            $ 635 "A_sel_v≔A_VL1"
            global A_sel_v=A_VL1
            $ 636 "A_sel_v_end≔A_VL1_END"
            global A_sel_v_end=A_VL1_END
            $ 637 "b2_par_cd≔0"
            global b2_par_cd=0
            $ 638 "If b1_cell_info_L≟A or b1_cell_info_L≟C or b1_cell_info_L≟c"
            if (b1_cell_info_L == A  or  b1_cell_info_L == C  or  b1_cell_info_L == c):
              $ 639 "Scallup_check≔ True "
              global Scallup_check=  True
            else:
              $ 640 "Else" "noBreak"
              $ 641 "Scallup_check≔ False "
              global Scallup_check=  False
            end
            $ 642 "Call MoveandTouchFun_3f"
            MoveandTouchFun_3f()
            $ 643 "If b1_cell_info_L≟A or b1_cell_info_L≟C or b1_cell_info_L≟c"
            if (b1_cell_info_L == A  or  b1_cell_info_L == C  or  b1_cell_info_L == c):
              $ 644 "If A_Prepos_l[A_HOR]≟p[0,0,0,0,0,0]"
              if (A_Prepos_l[A_HOR] == p[0,0,0,0,0,0]):
                $ 645 "direction(p[0,0,0,0,0,0],[0,-1,0],8,120,160)"
                direction(p[0,0,0,0,0,0],[0,-1,0],8,120,160)
                $ 647 "AAgcp≔get_actual_tcp_pose()"
                global AAgcp= get_actual_tcp_pose ()
                $ 648 "AAgangle≔up_left"
                global AAgangle=p[.492775857339, .409517380626, -.029063830209, -2.419264859926, -.998084331190, -1.368689080860]
                $ 649 "AAgtp≔p[AAgcp[0],AAgcp[1],AAgcp[2],AAgangle[3],AAgangle[4],AAgangle[5]]"
                global AAgtp=p[AAgcp[0],AAgcp[1],AAgcp[2],AAgangle[3],AAgangle[4],AAgangle[5]]
                $ 650 "MoveL"
                $ 651 "AAgtp" "breakAfter"
                movel(pose_trans(Base, AAgtp), a=0.08, v=0.08)
                $ 653 "for_z_VL1≔contact_fun(p[0,0,0,0,0,0],[0,0,-1],10000,15,15,  False)"
                global for_z_VL1=contact_fun(p[0,0,0,0,0,0],[0,0,-1],10000,15,15,  False)
                $ 654 "direction(p[0,0,0,0,0,0],[0,0,1],20,120,160)"
                direction(p[0,0,0,0,0,0],[0,0,1],20,120,160)
                $ 655 "write_welder(4, False )"
                write_welder(4,  False  )
              else:
                $ 656 "Else" "noBreak"
                $ 657 "for_z_VL1≔p[0,0,0,0,0,0]"
                global for_z_VL1=p[0,0,0,0,0,0]
              end
            end
            $ 658 "If top_touch_3f"
            if (top_touch_3f):
              $ 659 "touch_3f_up"
              $ 660 "b_touch_pos≔pose_add(A_Prepos_l[A_VL1], p[0,0,a8_wv_distance/1000,0,0,0])"
              global b_touch_pos= pose_add (A_Prepos_l[A_VL1], p[0,0,a8_wv_distance/1000,0,0,0])
              $ 661 "b_touch_pos≔tilt_3f_fun(b_touch_pos,[0,0],a5_f_hole[1])"
              global b_touch_pos=tilt_3f_fun(b_touch_pos,[0,0],a5_f_hole[1])
              $ 662 "MoveL"
              $ 663 "b_touch_pos" "breakAfter"
              movel(pose_trans(Base, b_touch_pos), a=0.35, v=0.35)
              $ 664 "touch_result≔touch_fun2(b_touch_pos,b2_left_par,b9_touch_sens)"
              global touch_result=touch_fun2(b_touch_pos,b2_left_par,b9_touch_sens)
              $ 665 "A_Touch_p[A_sel_v_end]=touch_result"
              A_Touch_p[A_sel_v_end]=touch_result
              $ 666 "If EXT_flag1[3]≟ True "
              if (EXT_flag1[3] ==   True  ):
                $ 667 "MoveL"
                $ 668 "manual_tp≔A_Touch_p[A_sel_v_end]"
                global manual_tp=A_Touch_p[A_sel_v_end]
                $ 669 "manual_tp≔tilt_3f_fun(A_Touch_p[A_sel_v_end],basic_tilt_3f,0)"
                global manual_tp=tilt_3f_fun(A_Touch_p[A_sel_v_end],basic_tilt_3f,0)
                $ 670 "manual_tp≔pose_trans(manual_tp, p[0,0,-10/1000,0,0,0])"
                global manual_tp= pose_trans (manual_tp, p[0,0,-10/1000,0,0,0])
                $ 671 "manual_tp" "breakAfter"
                movel(pose_trans(Base, manual_tp), a=0.3, v=0.15)
                $ 672 "Wait: 1.5"
                sleep(1.5)
              end
            end
          end
          $ 673 "HOR_ML"
          $ 674 "If A_Prepos_l[A_HOR_ML]≠p[0,0,0,0,0,0]"
          if (A_Prepos_l[A_HOR_ML] != p[0,0,0,0,0,0]):
            $ 675 "b2_left_par≔ True "
            global b2_left_par=  True
            $ 676 "b8_wv_2f≔ True "
            global b8_wv_2f=  True
            $ 677 "b7_tilt_degree≔[0,0,0]"
            global b7_tilt_degree=[0,0,0]
            $ 678 "A_sel_v≔A_HOR_ML"
            global A_sel_v=A_HOR_ML
            $ 679 "If b1_cell_info_L≟C or b1_cell_info_L≟D"
            if (b1_cell_info_L == C  or  b1_cell_info_L == D):
              $ 680 "wv_direction≔1"
              global wv_direction=1
              $ 681 "Call MoveFun"
              MoveFun()
              $ 682 "for_cal_xy≔contact_fun(p[0,0,0,0,0,0],[1,0,0],20000,20,20)"
              global for_cal_xy=contact_fun(p[0,0,0,0,0,0],[1,0,0],20000,20,20)
              $ 683 "direction(p[0,0,0,0,0,0],[-1,0,0],15,120,160)"
              direction(p[0,0,0,0,0,0],[-1,0,0],15,120,160)
              $ 684 "direction(p[0,0,0,0,0,0],[0,-1,0],60,120,160)"
              direction(p[0,0,0,0,0,0],[0,-1,0],60,120,160)
              $ 685 "direction(p[0,0,0,0,0,0],[1,0,0],20,120,160)"
              direction(p[0,0,0,0,0,0],[1,0,0],20,120,160)
              $ 686 "for_cal_x_wel≔contact_fun(p[0,0,0,0,0,0],[0,1,0],20000,20,20)"
              global for_cal_x_wel=contact_fun(p[0,0,0,0,0,0],[0,1,0],20000,20,20)
              $ 687 "direction(p[0,0,0,0,0,0],[0,-1,0],20,120,160)"
              direction(p[0,0,0,0,0,0],[0,-1,0],20,120,160)
              $ 688 "for_cal_y_wel≔contact_fun(p[0,0,0,0,0,0],[1,0,0],20000,20,20)"
              global for_cal_y_wel=contact_fun(p[0,0,0,0,0,0],[1,0,0],20000,20,20)
              $ 689 "direction(p[0,0,0,0,0,0],[-1,0,0],20,120,160)"
              direction(p[0,0,0,0,0,0],[-1,0,0],20,120,160)
              $ 690 "for_z_VLR2≔contact_fun(p[0,0,0,0,0,0],[0,0,-1],20000,20,20)"
              global for_z_VLR2=contact_fun(p[0,0,0,0,0,0],[0,0,-1],20000,20,20)
              $ 691 "direction(p[0,0,0,0,0,0],[0,0,1],20,120,160)"
              direction(p[0,0,0,0,0,0],[0,0,1],20,120,160)
              $ 692 "for_cal_rot≔A_Touch_p[A_HOR]"
              global for_cal_rot=A_Touch_p[A_HOR]
              $ 693 "A_Touch_p[A_sel_v]=p[for_cal_xy[0],for_cal_xy[1],for_z_VLR2[2],for_cal_rot[3],for_cal_rot[4],for_cal_rot[5]]"
              A_Touch_p[A_sel_v]=p[for_cal_xy[0],for_cal_xy[1],for_z_VLR2[2],for_cal_rot[3],for_cal_rot[4],for_cal_rot[5]]
              $ 694 "A_Touch_p[A_sel_v]=pose_trans(A_Touch_p[A_sel_v], p[Touch_dis/1000,0,0,0,0,0])"
              A_Touch_p[A_sel_v]= pose_trans (A_Touch_p[A_sel_v], p[Touch_dis/1000,0,0,0,0,0])
              $ 695 "write_welder(4, False )"
              write_welder(4,  False  )
            else:
              $ 696 "Else" "noBreak"
              $ 697 "wv_direction≔1"
              global wv_direction=1
              $ 698 "for_cal_rot≔A_Touch_p[A_HOR]"
              global for_cal_rot=A_Touch_p[A_HOR]
              $ 699 "Call MoveFun_cd"
              MoveFun_cd()
              $ 700 "for_cal_y_wel≔contact_fun(p[0,0,0,0,0,0],[1,0,0],20000,20,20)"
              global for_cal_y_wel=contact_fun(p[0,0,0,0,0,0],[1,0,0],20000,20,20)
              $ 701 "for_cal_y_wel[2]=for_cal_rot[2]"
              for_cal_y_wel[2]=for_cal_rot[2]
              $ 702 "dir_x_cal≔get_feature_Line(for_cal_rot,for_cal_y_wel)"
              global dir_x_cal=get_feature_Line(for_cal_rot,for_cal_y_wel)
              $ 703 "direction(p[0,0,0,0,0,0],[-1,0,0],40,120,160)"
              direction(p[0,0,0,0,0,0],[-1,0,0],40,120,160)
              $ 704 "direction(p[0,0,0,0,0,0],[0,-1,0],80,120,160)"
              direction(p[0,0,0,0,0,0],[0,-1,0],80,120,160)
              $ 705 "for_cal_y_wel≔contact_fun(p[0,0,0,0,0,0],[1,0,0],20000,20,20)"
              global for_cal_y_wel=contact_fun(p[0,0,0,0,0,0],[1,0,0],20000,20,20)
              $ 706 "direction(p[0,0,0,0,0,0],[-1,0,0],5,120,160)"
              direction(p[0,0,0,0,0,0],[-1,0,0],5,120,160)
              $ 707 "direction(p[0,0,0,0,0,0],[0,1,0],60,120,160)"
              direction(p[0,0,0,0,0,0],[0,1,0],60,120,160)
              $ 708 "direction(p[0,0,0,0,0,0],[1,0,0],7,120,160)"
              direction(p[0,0,0,0,0,0],[1,0,0],7,120,160)
              $ 709 "for_cal_x_wel≔contact_fun(p[0,0,0,0,0,0],[0,-1,0],20000,20,20)"
              global for_cal_x_wel=contact_fun(p[0,0,0,0,0,0],[0,-1,0],20000,20,20)
              $ 710 "get_ml≔get_feature_pose(for_cal_x_wel,for_cal_rot)"
              global get_ml=get_feature_pose(for_cal_x_wel,for_cal_rot)
              $ 712 "A_Touch_p[A_sel_v]=feature_offset(for_cal_rot,p[0,get_ml[0]+(-cd_offset+cd_extra_dis)/1000,0,0,0,0],dir_x_cal)"
              A_Touch_p[A_sel_v]=feature_offset(for_cal_rot,p[0,get_ml[0]+(-cd_offset+cd_extra_dis)/1000,0,0,0,0],dir_x_cal)
              $ 713 "direction(p[0,0,0,0,0,0],[0,1,0],5,120,160)"
              direction(p[0,0,0,0,0,0],[0,1,0],5,120,160)
              $ 714 "direction(p[0,0,0,0,0,0],[-1,0,0],20,120,160)"
              direction(p[0,0,0,0,0,0],[-1,0,0],20,120,160)
              $ 715 "write_welder(4, False )"
              write_welder(4,  False  )
            end
            $ 716 "homeing()"
            homeing()
          else:
            $ 717 "Else" "noBreak"
            $ 718 "homeing()"
            homeing()
          end
          $ 719 "VL2"
          $ 720 "If A_Prepos_l[A_VL2]≠p[0,0,0,0,0,0]"
          if (A_Prepos_l[A_VL2] != p[0,0,0,0,0,0]):
            $ 721 "b2_left_par≔ True "
            global b2_left_par=  True
            $ 722 "b8_wv_2f≔ False "
            global b8_wv_2f=  False
            $ 723 "b7_tilt_degree≔basic_tilt_3f"
            global b7_tilt_degree=basic_tilt_3f
            $ 724 "A_sel_v≔A_VL2"
            global A_sel_v=A_VL2
            $ 725 "A_sel_v_end≔A_VL2_END"
            global A_sel_v_end=A_VL2_END
            $ 726 "b2_par_cd≔1"
            global b2_par_cd=1
            $ 727 "If b1_cell_info_L≟A or b1_cell_info_L≟C or b1_cell_info_L≟c"
            if (b1_cell_info_L == A  or  b1_cell_info_L == C  or  b1_cell_info_L == c):
              $ 728 "Scallup_check≔ True "
              global Scallup_check=  True
            else:
              $ 729 "Else" "noBreak"
              $ 730 "Scallup_check≔ False "
              global Scallup_check=  False
            end
            $ 731 "If b1_cell_info_L≟d or b1_cell_info_L≟c"
            if (b1_cell_info_L == d  or  b1_cell_info_L == c):
              $ 732 "Halt"
              halt
            else:
              $ 733 "Else" "noBreak"
              $ 734 "If A_Touch_p[A_VL1]≟p[0,0,0,0,0,0]"
              if (A_Touch_p[A_VL1] == p[0,0,0,0,0,0]):
                $ 735 "Call MoveandTouchFun_3f"
                MoveandTouchFun_3f()
                $ 736 "If A_Prepos_l[A_HOR_ML]≟p[0,0,0,0,0,0]"
                if (A_Prepos_l[A_HOR_ML] == p[0,0,0,0,0,0]):
                  $ 737 "direction(p[0,0,0,0,0,0],[-1,-1,0],8,120,160)"
                  direction(p[0,0,0,0,0,0],[-1,-1,0],8,120,160)
                  $ 738 "AAgcp≔get_actual_tcp_pose()"
                  global AAgcp= get_actual_tcp_pose ()
                  $ 739 "AAgangle≔up_left"
                  global AAgangle=p[.492775857339, .409517380626, -.029063830209, -2.419264859926, -.998084331190, -1.368689080860]
                  $ 740 "AAgtp≔p[AAgcp[0],AAgcp[1],AAgcp[2],AAgangle[3],AAgangle[4],AAgangle[5]]"
                  global AAgtp=p[AAgcp[0],AAgcp[1],AAgcp[2],AAgangle[3],AAgangle[4],AAgangle[5]]
                  $ 741 "MoveL"
                  $ 742 "AAgtp" "breakAfter"
                  movel(pose_trans(Base, AAgtp), a=0.08, v=0.08)
                  $ 744 "for_z_VLR2≔contact_fun(p[0,0,0,0,0,0],[0,0,-1],20000,20,20)"
                  global for_z_VLR2=contact_fun(p[0,0,0,0,0,0],[0,0,-1],20000,20,20)
                  $ 745 "direction(p[0,0,0,0,0,0],[0,0,1],10,120,160)"
                  direction(p[0,0,0,0,0,0],[0,0,1],10,120,160)
                end
                $ 746 "touch_tmp≔A_Touch_p[A_sel_v]"
                global touch_tmp=A_Touch_p[A_sel_v]
                $ 747 "touch_tmp[2]=for_z_VLR2[2]"
                touch_tmp[2]=for_z_VLR2[2]
                $ 748 "A_Touch_p[A_sel_v]=touch_tmp"
                A_Touch_p[A_sel_v]=touch_tmp
                $ 749 "for_cal_y_wel≔A_Touch_p[A_sel_v]"
                global for_cal_y_wel=A_Touch_p[A_sel_v]
                $ 750 "for_cal_x_wel≔A_Touch_p[A_sel_v]"
                global for_cal_x_wel=A_Touch_p[A_sel_v]
              else:
                $ 751 "Else" "noBreak"
                $ 752 "If A_Prepos_l[A_HOR_ML]≟p[0,0,0,0,0,0]"
                if (A_Prepos_l[A_HOR_ML] == p[0,0,0,0,0,0]):
                  $ 753 "Call MoveFun"
                  MoveFun()
                  $ 754 "for_cal_y_wel≔contact_fun(p[0,0,0,0,0,0],[1,0,0],20000,20,20)"
                  global for_cal_y_wel=contact_fun(p[0,0,0,0,0,0],[1,0,0],20000,20,20)
                  $ 755 "direction(p[0,0,0,0,0,0],[-1,0,0],40,120,160)"
                  direction(p[0,0,0,0,0,0],[-1,0,0],40,120,160)
                  $ 756 "direction(p[0,0,0,0,0,0],[0,1,0],60,120,160)"
                  direction(p[0,0,0,0,0,0],[0,1,0],60,120,160)
                  $ 757 "var_2≔contact_fun(p[0,0,0,0,0,0],[1,0,0],20000,20,20)"
                  global var_2=contact_fun(p[0,0,0,0,0,0],[1,0,0],20000,20,20)
                  $ 758 "direction(p[0,0,0,0,0,0],[-1,0,0],5,120,160)"
                  direction(p[0,0,0,0,0,0],[-1,0,0],5,120,160)
                  $ 759 "direction(p[0,0,0,0,0,0],[0,-1,0],60,120,160)"
                  direction(p[0,0,0,0,0,0],[0,-1,0],60,120,160)
                  $ 760 "direction(p[0,0,0,0,0,0],[1,0,0],10,120,160)"
                  direction(p[0,0,0,0,0,0],[1,0,0],10,120,160)
                  $ 761 "for_cal_x_wel≔contact_fun(p[0,0,0,0,0,0],[0,1,0],20000,20,20)"
                  global for_cal_x_wel=contact_fun(p[0,0,0,0,0,0],[0,1,0],20000,20,20)
                  $ 762 "direction(p[0,0,0,0,0,0],[0,-1,0],20,120,160)"
                  direction(p[0,0,0,0,0,0],[0,-1,0],20,120,160)
                  $ 763 "AAgcp≔get_actual_tcp_pose()"
                  global AAgcp= get_actual_tcp_pose ()
                  $ 764 "AAgangle≔up_left"
                  global AAgangle=p[.492775857339, .409517380626, -.029063830209, -2.419264859926, -.998084331190, -1.368689080860]
                  $ 765 "AAgtp≔p[AAgcp[0],AAgcp[1],AAgcp[2],AAgangle[3],AAgangle[4],AAgangle[5]]"
                  global AAgtp=p[AAgcp[0],AAgcp[1],AAgcp[2],AAgangle[3],AAgangle[4],AAgangle[5]]
                  $ 766 "MoveL"
                  $ 767 "AAgtp" "breakAfter"
                  movel(pose_trans(Base, AAgtp), a=0.08, v=0.08)
                  $ 769 "for_z_VLR2≔contact_fun(p[0,0,0,0,0,0],[0,0,-1],20000,20,20)"
                  global for_z_VLR2=contact_fun(p[0,0,0,0,0,0],[0,0,-1],20000,20,20)
                  $ 770 "direction(p[0,0,0,0,0,0],[0,0,1],10,120,160)"
                  direction(p[0,0,0,0,0,0],[0,0,1],10,120,160)
                  $ 771 "direction(p[0,0,0,0,0,0],[-1,0,0],20,120,160)"
                  direction(p[0,0,0,0,0,0],[-1,0,0],20,120,160)
                end
                $ 772 "for_cal_rot≔A_Touch_p[A_VL1]"
                global for_cal_rot=A_Touch_p[A_VL1]
                $ 773 "touch_tmp=p[for_cal_y_wel[0],for_cal_x_wel[1],for_cal_x_wel[2],for_cal_rot[3],for_cal_rot[4],for_cal_rot[5]]"
                touch_tmp=p[for_cal_y_wel[0],for_cal_x_wel[1],for_cal_x_wel[2],for_cal_rot[3],for_cal_rot[4],for_cal_rot[5]]
                $ 774 "If Scallup_check≟ False "
                if (Scallup_check ==   False  ):
                  $ 775 "touch_tmp≔pose_trans(touch_tmp,p[-(Touch_dis)/1000,0,0,0,0,0])"
                  global touch_tmp= pose_trans (touch_tmp,p[-(Touch_dis)/1000,0,0,0,0,0])
                else:
                  $ 776 "Else" "noBreak"
                  $ 777 "Scallup_check≔ False "
                  global Scallup_check=  False
                end
                $ 778 "A_Touch_p[A_sel_v]=touch_tmp"
                A_Touch_p[A_sel_v]=touch_tmp
                $ 779 "write_welder(4, False )"
                write_welder(4,  False  )
              end
            end
            $ 780 "b2_par_cd≔0"
            global b2_par_cd=0
            $ 781 "homeing()"
            homeing()
          else:
            $ 782 "Else" "noBreak"
            $ 783 "homeing()"
            homeing()
          end
          $ 784 "HOR_R"
          $ 785 "If A_Prepos_l[A_HOR_R]≠p[0,0,0,0,0,0]"
          if (A_Prepos_l[A_HOR_R] != p[0,0,0,0,0,0]):
            $ 786 "b2_left_par≔ False "
            global b2_left_par=  False
            $ 787 "b8_wv_2f≔ True "
            global b8_wv_2f=  True
            $ 788 "b7_tilt_degree≔[0,0,0]"
            global b7_tilt_degree=[0,0,0]
            $ 789 "A_sel_v≔A_HOR_R"
            global A_sel_v=A_HOR_R
            $ 790 "wv_direction≔-1"
            global wv_direction=-1
            $ 791 "Call MoveandTouchFun_2f"
            MoveandTouchFun_2f()
            $ 793 "If b1_cell_info_R≟A or b1_cell_info_R≟C or b1_cell_info_R≟c"
            if (b1_cell_info_R == A  or  b1_cell_info_R == C  or  b1_cell_info_R == c):
              $ 794 "If A_Prepos_l[A_VR1]≟p[0,0,0,0,0,0]"
              if (A_Prepos_l[A_VR1] == p[0,0,0,0,0,0]):
                $ 796 "g_tp≔A_Prepos_l[A_HOR_R]"
                global g_tp=A_Prepos_l[A_HOR_R]
                $ 797 "Folder"
                $ 798 "g_cp≔get_actual_tcp_pose()"
                global g_cp= get_actual_tcp_pose ()
                $ 799 "g_cp≔pose_trans(g_cp, p[0,0,0,d2r(-12),d2r(5),0])"
                global g_cp= pose_trans (g_cp, p[0,0,0,d2r(-12),d2r(5),0])
                $ 800 "MoveL"
                $ 801 "g_cp" "breakAfter"
                movel(pose_trans(Base, g_cp), a=0.08, v=0.08)
                $ 804 "for_x_HOR_R≔contact_fun(A_Touch_p[A_HOR_R],[-1*wv_direction,0,0],10000,15,15,  False)"
                global for_x_HOR_R=contact_fun(A_Touch_p[A_HOR_R],[-1*wv_direction,0,0],10000,15,15,  False)
                $ 805 "direction(p[0,0,0,0,0,0],[0,1,0],20,120,160)"
                direction(p[0,0,0,0,0,0],[0,1,0],20,120,160)
                $ 806 "write_welder(4, False )"
                write_welder(4,  False  )
              else:
                $ 807 "Else" "noBreak"
                $ 808 "for_x_HOR_R≔p[0,0,0,0,0,0]"
                global for_x_HOR_R=p[0,0,0,0,0,0]
              end
            end
            $ 809 "wv_direction≔1"
            global wv_direction=1
            $ 810 "If point_dist(A_Prepos_l[A_HOR_R], A_Prepos_l[A_VR1])>0.0327"
            if (point_dist(A_Prepos_l[A_HOR_R], A_Prepos_l[A_VR1])>0.0327):
              $ 811 "homeing()"
              homeing()
            end
          end
          $ 812 "VR1"
          $ 813 "If A_Prepos_l[A_VR1]≠p[0,0,0,0,0,0]"
          if (A_Prepos_l[A_VR1] != p[0,0,0,0,0,0]):
            $ 814 "b2_left_par≔ False "
            global b2_left_par=  False
            $ 815 "b8_wv_2f≔ False "
            global b8_wv_2f=  False
            $ 816 "b7_tilt_degree≔basic_tilt_3f"
            global b7_tilt_degree=basic_tilt_3f
            $ 817 "A_sel_v≔A_VR1"
            global A_sel_v=A_VR1
            $ 818 "A_sel_v_end≔A_VR1_END"
            global A_sel_v_end=A_VR1_END
            $ 819 "b2_par_cd≔0"
            global b2_par_cd=0
            $ 820 "If b1_cell_info_R≟A or b1_cell_info_R≟C or b1_cell_info_R≟c"
            if (b1_cell_info_R == A  or  b1_cell_info_R == C  or  b1_cell_info_R == c):
              $ 821 "Scallup_check≔ True "
              global Scallup_check=  True
            else:
              $ 822 "Else" "noBreak"
              $ 823 "Scallup_check≔ False "
              global Scallup_check=  False
            end
            $ 824 "Call MoveandTouchFun_3f"
            MoveandTouchFun_3f()
            $ 825 "If b1_cell_info_R≟A or b1_cell_info_R≟C or b1_cell_info_R≟c"
            if (b1_cell_info_R == A  or  b1_cell_info_R == C  or  b1_cell_info_R == c):
              $ 826 "If A_Prepos_l[A_HOR_R]≟p[0,0,0,0,0,0]"
              if (A_Prepos_l[A_HOR_R] == p[0,0,0,0,0,0]):
                $ 827 "direction(p[0,0,0,0,0,0],[0,1,0],8,120,160)"
                direction(p[0,0,0,0,0,0],[0,1,0],8,120,160)
                $ 828 "AAgcp≔get_actual_tcp_pose()"
                global AAgcp= get_actual_tcp_pose ()
                $ 829 "AAgangle≔up_right"
                global AAgangle=p[.445203173045, -.406687378356, -.031125942276, 2.308490741423, -1.066468937023, 1.322151316133]
                $ 830 "AAgtp≔p[AAgcp[0],AAgcp[1],AAgcp[2],AAgangle[3],AAgangle[4],AAgangle[5]]"
                global AAgtp=p[AAgcp[0],AAgcp[1],AAgcp[2],AAgangle[3],AAgangle[4],AAgangle[5]]
                $ 831 "MoveL"
                $ 832 "AAgtp" "breakAfter"
                movel(pose_trans(Base, AAgtp), a=0.08, v=0.08)
                $ 834 "for_z_VR1≔contact_fun(p[0,0,0,0,0,0],[0,0,-1],10000,15,15,  False)"
                global for_z_VR1=contact_fun(p[0,0,0,0,0,0],[0,0,-1],10000,15,15,  False)
                $ 835 "direction(p[0,0,0,0,0,0],[0,0,1],20,120,160)"
                direction(p[0,0,0,0,0,0],[0,0,1],20,120,160)
                $ 836 "write_welder(4, False )"
                write_welder(4,  False  )
              else:
                $ 837 "Else" "noBreak"
                $ 838 "for_z_VR1≔p[0,0,0,0,0,0]"
                global for_z_VR1=p[0,0,0,0,0,0]
              end
            end
          end
          $ 839 "HOR_MR"
          $ 840 "If A_Prepos_l[A_HOR_MR]≠p[0,0,0,0,0,0]"
          if (A_Prepos_l[A_HOR_MR] != p[0,0,0,0,0,0]):
            $ 841 "INIT"
            $ 842 "b2_left_par≔ False "
            global b2_left_par=  False
            $ 843 "b8_wv_2f≔ True "
            global b8_wv_2f=  True
            $ 844 "b7_tilt_degree≔[0,0,0]"
            global b7_tilt_degree=[0,0,0]
            $ 845 "A_sel_v≔A_HOR_MR"
            global A_sel_v=A_HOR_MR
            $ 846 "If b1_cell_info_R≟C or b1_cell_info_R≟D"
            if (b1_cell_info_R == C  or  b1_cell_info_R == D):
              $ 847 "wv_direction≔-1"
              global wv_direction=-1
              $ 848 "Call MoveFun_cd"
              MoveFun_cd()
              $ 849 "for_cal_xy≔contact_fun(p[0,0,0,0,0,0],[1,0,0],20000,20,20)"
              global for_cal_xy=contact_fun(p[0,0,0,0,0,0],[1,0,0],20000,20,20)
              $ 850 "direction(p[0,0,0,0,0,0],[-1,0,0],15,120,160)"
              direction(p[0,0,0,0,0,0],[-1,0,0],15,120,160)
              $ 851 "direction(p[0,0,0,0,0,0],[0,1,0],60,120,160)"
              direction(p[0,0,0,0,0,0],[0,1,0],60,120,160)
              $ 852 "direction(p[0,0,0,0,0,0],[1,0,0],20,120,160)"
              direction(p[0,0,0,0,0,0],[1,0,0],20,120,160)
              $ 853 "for_cal_x_wel≔contact_fun(p[0,0,0,0,0,0],[0,-1,0],20000,20,20)"
              global for_cal_x_wel=contact_fun(p[0,0,0,0,0,0],[0,-1,0],20000,20,20)
              $ 854 "direction(p[0,0,0,0,0,0],[0,1,0],20,120,160)"
              direction(p[0,0,0,0,0,0],[0,1,0],20,120,160)
              $ 855 "for_cal_y_wel≔contact_fun(p[0,0,0,0,0,0],[1,0,0],20000,20,20)"
              global for_cal_y_wel=contact_fun(p[0,0,0,0,0,0],[1,0,0],20000,20,20)
              $ 856 "direction(p[0,0,0,0,0,0],[-1,0,0],8,120,160)"
              direction(p[0,0,0,0,0,0],[-1,0,0],8,120,160)
              $ 857 "for_cal_zr≔contact_fun(p[0,0,0,0,0,0],[0,0,-1],20000,20,20)"
              global for_cal_zr=contact_fun(p[0,0,0,0,0,0],[0,0,-1],20000,20,20)
              $ 858 "direction(p[0,0,0,0,0,0],[0,0,1],20,120,160)"
              direction(p[0,0,0,0,0,0],[0,0,1],20,120,160)
              $ 859 "for_cal_rot≔A_Touch_p[A_HOR_R]"
              global for_cal_rot=A_Touch_p[A_HOR_R]
              $ 860 "A_Touch_p[A_sel_v]=p[for_cal_xy[0],for_cal_xy[1],for_cal_zr[2],for_cal_rot[3],for_cal_rot[4],for_cal_rot[5]]"
              A_Touch_p[A_sel_v]=p[for_cal_xy[0],for_cal_xy[1],for_cal_zr[2],for_cal_rot[3],for_cal_rot[4],for_cal_rot[5]]
              $ 861 "A_Touch_p[A_sel_v]=pose_trans(A_Touch_p[A_sel_v], p[-Touch_dis/1000,0,0,0,0,0])"
              A_Touch_p[A_sel_v]= pose_trans (A_Touch_p[A_sel_v], p[-Touch_dis/1000,0,0,0,0,0])
              $ 862 "write_welder(4, False )"
              write_welder(4,  False  )
            else:
              $ 863 "Else" "noBreak"
              $ 864 "wv_direction≔-1"
              global wv_direction=-1
              $ 865 "for_cal_rot≔A_Touch_p[A_HOR_R]"
              global for_cal_rot=A_Touch_p[A_HOR_R]
              $ 866 "Call MoveFun_cd"
              MoveFun_cd()
              $ 867 "for_cal_y_wel≔contact_fun(p[0,0,0,0,0,0],[1,0,0],20000,20,20)"
              global for_cal_y_wel=contact_fun(p[0,0,0,0,0,0],[1,0,0],20000,20,20)
              $ 868 "vr2_p1≔for_cal_y_wel"
              global vr2_p1=for_cal_y_wel
              $ 869 "for_cal_y_wel[2]=for_cal_rot[2]"
              for_cal_y_wel[2]=for_cal_rot[2]
              $ 870 "dir_x_cal≔get_feature_Line(for_cal_rot,for_cal_y_wel)"
              global dir_x_cal=get_feature_Line(for_cal_rot,for_cal_y_wel)
              $ 871 "vr2_p2≔feature_offset(vr2_p1,p[0,0.02,0,0,0,0],dir_x_cal)"
              global vr2_p2=feature_offset(vr2_p1,p[0,0.02,0,0,0,0],dir_x_cal)
              $ 872 "direction(p[0,0,0,0,0,0],[-1,0,0],40,120,160)"
              direction(p[0,0,0,0,0,0],[-1,0,0],40,120,160)
              $ 873 "direction(p[0,0,0,0,0,0],[0,1,0],80,120,160)"
              direction(p[0,0,0,0,0,0],[0,1,0],80,120,160)
              $ 874 "for_cal_y_wel≔contact_fun(p[0,0,0,0,0,0],[1,0,0],20000,20,20)"
              global for_cal_y_wel=contact_fun(p[0,0,0,0,0,0],[1,0,0],20000,20,20)
              $ 875 "direction(p[0,0,0,0,0,0],[-1,0,0],5,120,160)"
              direction(p[0,0,0,0,0,0],[-1,0,0],5,120,160)
              $ 876 "direction(p[0,0,0,0,0,0],[0,-1,0],60,120,160)"
              direction(p[0,0,0,0,0,0],[0,-1,0],60,120,160)
              $ 877 "direction(p[0,0,0,0,0,0],[1,0,0],7,120,160)"
              direction(p[0,0,0,0,0,0],[1,0,0],7,120,160)
              $ 878 "for_cal_x_wel≔contact_fun(p[0,0,0,0,0,0],[0,1,0],20000,20,20)"
              global for_cal_x_wel=contact_fun(p[0,0,0,0,0,0],[0,1,0],20000,20,20)
              $ 879 "vr2_p3≔for_cal_x_wel"
              global vr2_p3=for_cal_x_wel
              $ 880 "get_ml≔get_feature_pose(for_cal_x_wel,for_cal_rot)"
              global get_ml=get_feature_pose(for_cal_x_wel,for_cal_rot)
              $ 882 "A_Touch_p[A_sel_v]=feature_offset(for_cal_rot,p[0,-get_ml[0]+(-cd_offset+cd_extra_dis)/1000,0,0,0,0],dir_x_cal)"
              A_Touch_p[A_sel_v]=feature_offset(for_cal_rot,p[0,-get_ml[0]+(-cd_offset+cd_extra_dis)/1000,0,0,0,0],dir_x_cal)
              $ 883 "vr2_p4≔A_Touch_p[A_HOR_MR]"
              global vr2_p4=A_Touch_p[A_HOR_MR]
              $ 884 "direction(p[0,0,0,0,0,0],[0,-1,0],5,120,160)"
              direction(p[0,0,0,0,0,0],[0,-1,0],5,120,160)
              $ 885 "direction(p[0,0,0,0,0,0],[-1,0,0],20,120,160)"
              direction(p[0,0,0,0,0,0],[-1,0,0],20,120,160)
              $ 886 "write_welder(4, False )"
              write_welder(4,  False  )
            end
            $ 887 "homeing()"
            homeing()
            $ 888 "wv_direction≔1"
            global wv_direction=1
          else:
            $ 889 "Else" "noBreak"
            $ 890 "homeing()"
            homeing()
          end
          $ 891 "VR2"
          $ 892 "If A_Prepos_l[A_VR2]≠p[0,0,0,0,0,0]"
          if (A_Prepos_l[A_VR2] != p[0,0,0,0,0,0]):
            $ 893 "Init"
            $ 894 "b2_left_par≔ False "
            global b2_left_par=  False
            $ 895 "b8_wv_2f≔ False "
            global b8_wv_2f=  False
            $ 896 "b7_tilt_degree≔basic_tilt_3f"
            global b7_tilt_degree=basic_tilt_3f
            $ 897 "A_sel_v≔A_VR2"
            global A_sel_v=A_VR2
            $ 898 "A_sel_v_end≔A_VR2_END"
            global A_sel_v_end=A_VR2_END
            $ 899 "b2_par_cd≔1"
            global b2_par_cd=1
            $ 900 "If b1_cell_info_R≟A or b1_cell_info_R≟C or b1_cell_info_R≟c"
            if (b1_cell_info_R == A  or  b1_cell_info_R == C  or  b1_cell_info_R == c):
              $ 901 "Scallup_check≔ True "
              global Scallup_check=  True
            else:
              $ 902 "Else" "noBreak"
              $ 903 "Scallup_check≔ False "
              global Scallup_check=  False
            end
            $ 904 "If b1_cell_info_R≟d or b1_cell_info_R≟c"
            if (b1_cell_info_R == d  or  b1_cell_info_R == c):
              $ 905 "Halt"
              halt
              $ 906 "If vr2_p1≟p[0,0,0,0,0,0]"
              if (vr2_p1 == p[0,0,0,0,0,0]):
                $ 907 "Call MoveFun_cd"
                MoveFun_cd()
                $ 908 "vr2_p1≔contact_fun(p[0,0,0,0,0,0],[1,0,0],20000,20,20)"
                global vr2_p1=contact_fun(p[0,0,0,0,0,0],[1,0,0],20000,20,20)
                $ 909 "direction(p[0,0,0,0,0,0],[-1,0,0],20,120,160)"
                direction(p[0,0,0,0,0,0],[-1,0,0],20,120,160)
                $ 910 "direction(p[0,0,0,0,0,0],[0,1,0],10,120,160)"
                direction(p[0,0,0,0,0,0],[0,1,0],10,120,160)
                $ 911 "vr2_p2≔contact_fun(p[0,0,0,0,0,0],[1,0,0],20000,20,20)"
                global vr2_p2=contact_fun(p[0,0,0,0,0,0],[1,0,0],20000,20,20)
                $ 912 "direction(p[0,0,0,0,0,0],[-1,0,0],14,120,160)"
                direction(p[0,0,0,0,0,0],[-1,0,0],14,120,160)
                $ 913 "vr2_p3≔contact_fun(p[0,0,0,0,0,0],[0,1,0],20000,20,20)"
                global vr2_p3=contact_fun(p[0,0,0,0,0,0],[0,1,0],20000,20,20)
                $ 914 "direction(p[0,0,0,0,0,0],[0,-1,0],30,120,160)"
                direction(p[0,0,0,0,0,0],[0,-1,0],30,120,160)
                $ 915 "direction(p[0,0,0,0,0,0],[-1,0,0],20,120,160)"
                direction(p[0,0,0,0,0,0],[-1,0,0],20,120,160)
                $ 916 "vr2_p4≔contact_fun(p[0,0,0,0,0,0],[0,0,-1],20000,20,20)"
                global vr2_p4=contact_fun(p[0,0,0,0,0,0],[0,0,-1],20000,20,20)
                $ 917 "direction(p[0,0,0,0,0,0],[0,0,1],40,120,160)"
                direction(p[0,0,0,0,0,0],[0,0,1],40,120,160)
                $ 918 "A_Touch_p[A_sel_v]=touch_xyz_get_middle(vr2_p1,vr2_p2,vr2_p3,vr2_p4)"
                A_Touch_p[A_sel_v]=touch_xyz_get_middle(vr2_p1,vr2_p2,vr2_p3,vr2_p4)
                $ 919 "var_4≔A_Touch_p[A_sel_v]"
                global var_4=A_Touch_p[A_sel_v]
                $ 920 "var_4≔pose_trans(var_4, p[a6_callar_vert/1000,0,0,0,0,0])"
                global var_4= pose_trans (var_4, p[a6_callar_vert/1000,0,0,0,0,0])
                $ 921 "var_5≔get_actual_tcp_pose()"
                global var_5= get_actual_tcp_pose ()
                $ 922 "var_5[2]=var_4[2]"
                var_5[2]=var_4[2]
                $ 923 "var_5≔pose_trans(var_5, p[0,0,0,0,d2r(10),0])"
                global var_5= pose_trans (var_5, p[0,0,0,0,d2r(10),0])
                $ 924 "MoveL"
                $ 925 "var_5" "breakAfter"
                movel(pose_trans(Base, var_5), a=0.1, v=0.1)
                $ 926 "vr2_p1_up≔contact_fun(p[0,0,0,0,0,0],[1,0,0],20000,20,20)"
                global vr2_p1_up=contact_fun(p[0,0,0,0,0,0],[1,0,0],20000,20,20)
                $ 927 "direction(p[0,0,0,0,0,0],[-1,0,0],20,120,160)"
                direction(p[0,0,0,0,0,0],[-1,0,0],20,120,160)
                $ 928 "direction(p[0,0,0,0,0,0],[0,1,0],10,120,160)"
                direction(p[0,0,0,0,0,0],[0,1,0],10,120,160)
                $ 929 "vr2_p2_up≔contact_fun(p[0,0,0,0,0,0],[1,0,0],20000,20,20)"
                global vr2_p2_up=contact_fun(p[0,0,0,0,0,0],[1,0,0],20000,20,20)
                $ 930 "direction(p[0,0,0,0,0,0],[-1,0,0],14,120,160)"
                direction(p[0,0,0,0,0,0],[-1,0,0],14,120,160)
                $ 931 "vr2_p3_up≔contact_fun(p[0,0,0,0,0,0],[0,1,0],20000,20,20)"
                global vr2_p3_up=contact_fun(p[0,0,0,0,0,0],[0,1,0],20000,20,20)
                $ 932 "direction(p[0,0,0,0,0,0],[0,-1,0],30,120,160)"
                direction(p[0,0,0,0,0,0],[0,-1,0],30,120,160)
                $ 933 "direction(p[0,0,0,0,0,0],[-1,0,0],20,120,160)"
                direction(p[0,0,0,0,0,0],[-1,0,0],20,120,160)
              end
              $ 934 "A_Touch_p[A_sel_v+9]=touch_4point(vr2_p1_up,vr2_p2_up,vr2_p3_up)"
              A_Touch_p[A_sel_v+9]=touch_4point(vr2_p1_up,vr2_p2_up,vr2_p3_up)
              $ 935 "A_Touch_p[A_sel_v+9]=ori_pose(A_Touch_p[A_sel_v+9],A_Touch_p[A_sel_v])"
              A_Touch_p[A_sel_v+9]=ori_pose(A_Touch_p[A_sel_v+9],A_Touch_p[A_sel_v])
            else:
              $ 936 "Else" "noBreak"
              $ 937 "If A_Touch_p[A_VR1]≟p[0,0,0,0,0,0]"
              if (A_Touch_p[A_VR1] == p[0,0,0,0,0,0]):
                $ 938 "Call MoveandTouchFun_3f"
                MoveandTouchFun_3f()
                $ 939 "touch_tmp≔A_Touch_p[A_sel_v]"
                global touch_tmp=A_Touch_p[A_sel_v]
                $ 940 "If A_Prepos_l[A_HOR_MR]≟p[0,0,0,0,0,0]"
                if (A_Prepos_l[A_HOR_MR] == p[0,0,0,0,0,0]):
                  $ 941 "direction(p[0,0,0,0,0,0],[-1,1,0],8,120,160)"
                  direction(p[0,0,0,0,0,0],[-1,1,0],8,120,160)
                  $ 942 "AAgcp≔get_actual_tcp_pose()"
                  global AAgcp= get_actual_tcp_pose ()
                  $ 943 "AAgangle≔up_right"
                  global AAgangle=p[.445203173045, -.406687378356, -.031125942276, 2.308490741423, -1.066468937023, 1.322151316133]
                  $ 944 "AAgtp≔p[AAgcp[0],AAgcp[1],AAgcp[2],AAgangle[3],AAgangle[4],AAgangle[5]]"
                  global AAgtp=p[AAgcp[0],AAgcp[1],AAgcp[2],AAgangle[3],AAgangle[4],AAgangle[5]]
                  $ 945 "MoveL"
                  $ 946 "AAgtp" "breakAfter"
                  movel(pose_trans(Base, AAgtp), a=0.08, v=0.08)
                  $ 948 "for_z_VLR2≔contact_fun(p[0,0,0,0,0,0],[0,0,-1],20000,20,20)"
                  global for_z_VLR2=contact_fun(p[0,0,0,0,0,0],[0,0,-1],20000,20,20)
                  $ 949 "touch_tmp[2]=for_z_VLR2[2]"
                  touch_tmp[2]=for_z_VLR2[2]
                end
                $ 950 "A_Touch_p[A_sel_v]=touch_tmp"
                A_Touch_p[A_sel_v]=touch_tmp
                $ 951 "for_cal_y_wel≔A_Touch_p[A_sel_v]"
                global for_cal_y_wel=A_Touch_p[A_sel_v]
                $ 952 "for_cal_x_wel≔A_Touch_p[A_sel_v]"
                global for_cal_x_wel=A_Touch_p[A_sel_v]
              else:
                $ 953 "Else" "noBreak"
                $ 954 "If A_Prepos_l[A_HOR_MR]≟p[0,0,0,0,0,0]"
                if (A_Prepos_l[A_HOR_MR] == p[0,0,0,0,0,0]):
                  $ 955 "Call MoveFun"
                  MoveFun()
                  $ 956 "for_cal_y_wel≔contact_fun(p[0,0,0,0,0,0],[1,0,0],20000,20,20)"
                  global for_cal_y_wel=contact_fun(p[0,0,0,0,0,0],[1,0,0],20000,20,20)
                  $ 957 "direction(p[0,0,0,0,0,0],[-1,0,0],40,120,160)"
                  direction(p[0,0,0,0,0,0],[-1,0,0],40,120,160)
                  $ 958 "direction(p[0,0,0,0,0,0],[0,-1,0],60,120,160)"
                  direction(p[0,0,0,0,0,0],[0,-1,0],60,120,160)
                  $ 959 "var_2≔contact_fun(p[0,0,0,0,0,0],[1,0,0],20000,20,20)"
                  global var_2=contact_fun(p[0,0,0,0,0,0],[1,0,0],20000,20,20)
                  $ 960 "direction(p[0,0,0,0,0,0],[-1,0,0],5,120,160)"
                  direction(p[0,0,0,0,0,0],[-1,0,0],5,120,160)
                  $ 961 "direction(p[0,0,0,0,0,0],[0,1,0],60,120,160)"
                  direction(p[0,0,0,0,0,0],[0,1,0],60,120,160)
                  $ 962 "direction(p[0,0,0,0,0,0],[1,0,0],10,120,160)"
                  direction(p[0,0,0,0,0,0],[1,0,0],10,120,160)
                  $ 963 "for_cal_x_wel≔contact_fun(p[0,0,0,0,0,0],[0,-1,0],20000,20,20)"
                  global for_cal_x_wel=contact_fun(p[0,0,0,0,0,0],[0,-1,0],20000,20,20)
                  $ 964 "direction(p[0,0,0,0,0,0],[0,1,0],20,120,160)"
                  direction(p[0,0,0,0,0,0],[0,1,0],20,120,160)
                  $ 965 "AAgcp≔get_actual_tcp_pose()"
                  global AAgcp= get_actual_tcp_pose ()
                  $ 966 "AAgangle≔up_right"
                  global AAgangle=p[.445203173045, -.406687378356, -.031125942276, 2.308490741423, -1.066468937023, 1.322151316133]
                  $ 967 "AAgtp≔p[AAgcp[0],AAgcp[1],AAgcp[2],AAgangle[3],AAgangle[4],AAgangle[5]]"
                  global AAgtp=p[AAgcp[0],AAgcp[1],AAgcp[2],AAgangle[3],AAgangle[4],AAgangle[5]]
                  $ 968 "MoveL"
                  $ 969 "AAgtp" "breakAfter"
                  movel(pose_trans(Base, AAgtp), a=0.1, v=0.1)
                  $ 971 "for_z_VLR2≔contact_fun(p[0,0,0,0,0,0],[0,0,-1],20000,20,20)"
                  global for_z_VLR2=contact_fun(p[0,0,0,0,0,0],[0,0,-1],20000,20,20)
                  $ 972 "direction(p[0,0,0,0,0,0],[0,0,1],20,120,160)"
                  direction(p[0,0,0,0,0,0],[0,0,1],20,120,160)
                  $ 973 "direction(p[0,0,0,0,0,0],[-1,0,0],20,120,160)"
                  direction(p[0,0,0,0,0,0],[-1,0,0],20,120,160)
                end
                $ 974 "for_cal_rot≔A_Touch_p[A_VR1]"
                global for_cal_rot=A_Touch_p[A_VR1]
                $ 976 "touch_tmp=p[for_cal_y_wel[0],for_cal_x_wel[1],for_cal_x_wel[2],for_cal_rot[3],for_cal_rot[4],for_cal_rot[5]]"
                touch_tmp=p[for_cal_y_wel[0],for_cal_x_wel[1],for_cal_x_wel[2],for_cal_rot[3],for_cal_rot[4],for_cal_rot[5]]
                $ 977 "If Scallup_check≟ False "
                if (Scallup_check ==   False  ):
                  $ 978 "touch_tmp≔pose_trans(touch_tmp,p[-(Touch_dis)/1000,0,0,0,0,0])"
                  global touch_tmp= pose_trans (touch_tmp,p[-(Touch_dis)/1000,0,0,0,0,0])
                else:
                  $ 979 "Else" "noBreak"
                  $ 980 "Scallup_check≔ False "
                  global Scallup_check=  False
                end
                $ 981 "A_Touch_p[A_sel_v]=touch_tmp"
                A_Touch_p[A_sel_v]=touch_tmp
                $ 982 "write_welder(4, False )"
                write_welder(4,  False  )
              end
            end
            $ 983 "b2_par_cd≔0"
            global b2_par_cd=0
            $ 984 "homeing()"
            homeing()
          else:
            $ 985 "Else" "noBreak"
            $ 986 "homeing()"
            homeing()
          end
          $ 987 "write_welder(4,False)"
          write_welder(4,False)
          $ 1044 "Touch After Offset"
          $ 1045 "touch_after_offset"
          $ 1046 "HOR"
          $ 1047 "If A_Prepos_l[A_HOR]≠p[0,0,0,0,0,0]"
          if (A_Prepos_l[A_HOR] != p[0,0,0,0,0,0]):
            $ 1048 "If b1_cell_info_L≟A or b1_cell_info_L≟C or b1_cell_info_L≟c"
            if (b1_cell_info_L == A  or  b1_cell_info_L == C  or  b1_cell_info_L == c):
              $ 1049 "If for_x_HOR≟p[0,0,0,0,0,0] and A_Touch_p[A_VL1]≠p[0,0,0,0,0,0]"
              if (for_x_HOR == p[0,0,0,0,0,0]  and  A_Touch_p[A_VL1] != p[0,0,0,0,0,0]):
                $ 1050 "for_x_HOR≔A_Touch_p[A_VL1]"
                global for_x_HOR=A_Touch_p[A_VL1]
              end
              $ 1051 "If for_x_HOR≠p[0,0,0,0,0,0]"
              if (for_x_HOR != p[0,0,0,0,0,0]):
                $ 1052 "x_diff≔get_feature_pose(for_x_HOR,A_Touch_p[A_HOR])"
                global x_diff=get_feature_pose(for_x_HOR,A_Touch_p[A_HOR])
                $ 1053 "A_Touch_p[A_HOR]=pose_trans(A_Touch_p[A_HOR], p[x_diff[0],0,0,0,0,0])"
                A_Touch_p[A_HOR]= pose_trans (A_Touch_p[A_HOR], p[x_diff[0],0,0,0,0,0])
                $ 1054 "If b1_cell_info_L≟B or b1_cell_info_L≟D or b1_cell_info_L≟d or b1_cell_info_L≟E or b1_cell_info_L≟e"
                if (b1_cell_info_L == B  or  b1_cell_info_L == D  or  b1_cell_info_L == d  or  b1_cell_info_L == E  or  b1_cell_info_L == e):
                  $ 1055 "A_Touch_p[A_HOR]=pose_trans(A_Touch_p[A_HOR], p[hor_l_scallup/1000,0,0,0,0,0])"
                  A_Touch_p[A_HOR]= pose_trans (A_Touch_p[A_HOR], p[hor_l_scallup/1000,0,0,0,0,0])
                end
              end
            end
            $ 1056 "A_Touch_p[A_HOR]=pose_trans(A_Touch_p[A_HOR], p[offset_2f_begin/1000,0,0,0,0,0])"
            A_Touch_p[A_HOR]= pose_trans (A_Touch_p[A_HOR], p[offset_2f_begin/1000,0,0,0,0,0])
          end
          $ 1057 "VL1"
          $ 1058 "If A_Prepos_l[A_VL1]≠p[0,0,0,0,0,0]"
          if (A_Prepos_l[A_VL1] != p[0,0,0,0,0,0]):
            $ 1059 "If b1_cell_info_L≟A or b1_cell_info_L≟C or b1_cell_info_L≟c"
            if (b1_cell_info_L == A  or  b1_cell_info_L == C  or  b1_cell_info_L == c):
              $ 1060 "'3f only does not apply offset'"
              # '3f only does not apply offset'
              $ 1061 "If for_z_VL1≟p[0,0,0,0,0,0] and A_Touch_p[A_HOR]≠p[0,0,0,0,0,0]"
              if (for_z_VL1 == p[0,0,0,0,0,0]  and  A_Touch_p[A_HOR] != p[0,0,0,0,0,0]):
                $ 1062 "for_z_VL1≔A_Touch_p[A_HOR]"
                global for_z_VL1=A_Touch_p[A_HOR]
              end
              $ 1063 "Comment"
              # Comment
              $ 1064 "If for_z_VL1≠p[0,0,0,0,0,0]"
              if (for_z_VL1 != p[0,0,0,0,0,0]):
                $ 1065 "z_diff≔get_feature_pose(for_z_VL1,A_Touch_p[A_VL1])"
                global z_diff=get_feature_pose(for_z_VL1,A_Touch_p[A_VL1])
                $ 1066 "A_Touch_p[A_VL1]=pose_trans(A_Touch_p[A_VL1], p[z_diff[0],0,0,0,0,0])"
                A_Touch_p[A_VL1]= pose_trans (A_Touch_p[A_VL1], p[z_diff[0],0,0,0,0,0])
              end
              $ 1067 "If b1_cell_info_L≟B or b1_cell_info_L≟D or b1_cell_info_L≟d or b1_cell_info_L≟E or b1_cell_info_L≟e"
              if (b1_cell_info_L == B  or  b1_cell_info_L == D  or  b1_cell_info_L == d  or  b1_cell_info_L == E  or  b1_cell_info_L == e):
                $ 1068 "A_Touch_p[A_VL1]=pose_trans(A_Touch_p[A_VL1], p[vert_scallup_l/1000,0,0,0,0,0])"
                A_Touch_p[A_VL1]= pose_trans (A_Touch_p[A_VL1], p[vert_scallup_l/1000,0,0,0,0,0])
              end
            end
            $ 1070 "A_Touch_p[A_VL1]=pose_trans(A_Touch_p[A_VL1], p[offset_3f_begin/1000,0,0,0,0,0])"
            A_Touch_p[A_VL1]= pose_trans (A_Touch_p[A_VL1], p[offset_3f_begin/1000,0,0,0,0,0])
          end
          $ 1071 "VL2"
          $ 1072 "If A_Prepos_l[A_VL2]≠p[0,0,0,0,0,0]"
          if (A_Prepos_l[A_VL2] != p[0,0,0,0,0,0]):
            $ 1073 "If b1_cell_info_L≟A or b1_cell_info_L≟C or b1_cell_info_L≟c or b1_cell_info_L≟D or b1_cell_info_L≟d or b1_cell_info_L≟E"
            if (b1_cell_info_L == A  or  b1_cell_info_L == C  or  b1_cell_info_L == c  or  b1_cell_info_L == D  or  b1_cell_info_L == d  or  b1_cell_info_L == E):
              $ 1074 "'3f only does not apply offset'"
              # '3f only does not apply offset'
              $ 1075 "If for_z_VLR2≟p[0,0,0,0,0,0] and A_Touch_p[A_HOR_ML]≠p[0,0,0,0,0,0]"
              if (for_z_VLR2 == p[0,0,0,0,0,0]  and  A_Touch_p[A_HOR_ML] != p[0,0,0,0,0,0]):
                $ 1076 "for_z_VLR2≔A_Touch_p[A_HOR_ML]"
                global for_z_VLR2=A_Touch_p[A_HOR_ML]
              end
              $ 1077 "Comment"
              # Comment
              $ 1078 "If for_z_VLR2≠p[0,0,0,0,0,0]"
              if (for_z_VLR2 != p[0,0,0,0,0,0]):
                $ 1079 "z_diff≔get_feature_pose(for_z_VLR2,A_Touch_p[A_VL2])"
                global z_diff=get_feature_pose(for_z_VLR2,A_Touch_p[A_VL2])
                $ 1080 "A_Touch_p[A_VL2]=pose_trans(A_Touch_p[A_VL2], p[z_diff[0],0,0,0,0,0])"
                A_Touch_p[A_VL2]= pose_trans (A_Touch_p[A_VL2], p[z_diff[0],0,0,0,0,0])
              end
              $ 1081 "If b1_cell_info_L≟E or b1_cell_info_L≟e"
              if (b1_cell_info_L == E  or  b1_cell_info_L == e):
                $ 1082 "A_Touch_p[A_VL2]=pose_trans(A_Touch_p[A_VL2], p[vert_scallup_l/1000,0,0,0,0,0])"
                A_Touch_p[A_VL2]= pose_trans (A_Touch_p[A_VL2], p[vert_scallup_l/1000,0,0,0,0,0])
              end
            end
            $ 1083 "A_Touch_p[A_VL2]=pose_trans(A_Touch_p[A_VL2], p[offset_3f_begin/1000,0,0,0,0,0])"
            A_Touch_p[A_VL2]= pose_trans (A_Touch_p[A_VL2], p[offset_3f_begin/1000,0,0,0,0,0])
          end
          $ 1084 "HOR_R"
          $ 1085 "If A_Prepos_l[A_HOR_R]≠p[0,0,0,0,0,0]"
          if (A_Prepos_l[A_HOR_R] != p[0,0,0,0,0,0]):
            $ 1086 "If b1_cell_info_R≟A or b1_cell_info_R≟C or b1_cell_info_R≟c"
            if (b1_cell_info_R == A  or  b1_cell_info_R == C  or  b1_cell_info_R == c):
              $ 1087 "If for_x_HOR_R≟p[0,0,0,0,0,0] and A_Touch_p[A_VR1]≠p[0,0,0,0,0,0]"
              if (for_x_HOR_R == p[0,0,0,0,0,0]  and  A_Touch_p[A_VR1] != p[0,0,0,0,0,0]):
                $ 1088 "for_x_HOR_R≔A_Touch_p[A_VR1]"
                global for_x_HOR_R=A_Touch_p[A_VR1]
              end
              $ 1089 "If for_x_HOR≠p[0,0,0,0,0,0]"
              if (for_x_HOR != p[0,0,0,0,0,0]):
                $ 1090 "x_diff≔get_feature_pose(for_x_HOR_R,A_Touch_p[A_HOR_R])"
                global x_diff=get_feature_pose(for_x_HOR_R,A_Touch_p[A_HOR_R])
                $ 1091 "A_Touch_p[A_HOR_R]=pose_trans(A_Touch_p[A_HOR_R], p[x_diff[0],0,0,0,0,0])"
                A_Touch_p[A_HOR_R]= pose_trans (A_Touch_p[A_HOR_R], p[x_diff[0],0,0,0,0,0])
                $ 1092 "If b1_cell_info_R≟B or b1_cell_info_R≟D or b1_cell_info_R≟d or b1_cell_info_R≟E or b1_cell_info_R≟e"
                if (b1_cell_info_R == B  or  b1_cell_info_R == D  or  b1_cell_info_R == d  or  b1_cell_info_R == E  or  b1_cell_info_R == e):
                  $ 1093 "A_Touch_p[A_HOR_R]=pose_trans(A_Touch_p[A_HOR_R], p[-hor_r_scallup/1000,0,0,0,0,0])"
                  A_Touch_p[A_HOR_R]= pose_trans (A_Touch_p[A_HOR_R], p[-hor_r_scallup/1000,0,0,0,0,0])
                end
              end
            end
            $ 1094 "A_Touch_p[A_HOR_R]=pose_trans(A_Touch_p[A_HOR_R], p[-offset_2f_begin/1000,0,0,0,0,0])"
            A_Touch_p[A_HOR_R]= pose_trans (A_Touch_p[A_HOR_R], p[-offset_2f_begin/1000,0,0,0,0,0])
          end
          $ 1095 "VR1"
          $ 1096 "If A_Prepos_l[A_VR1]≠p[0,0,0,0,0,0]"
          if (A_Prepos_l[A_VR1] != p[0,0,0,0,0,0]):
            $ 1097 "If b1_cell_info_R≟A or b1_cell_info_R≟C or b1_cell_info_R≟c"
            if (b1_cell_info_R == A  or  b1_cell_info_R == C  or  b1_cell_info_R == c):
              $ 1098 "If for_z_VR1≟p[0,0,0,0,0,0] and A_Touch_p[A_HOR_R]≠p[0,0,0,0,0,0]"
              if (for_z_VR1 == p[0,0,0,0,0,0]  and  A_Touch_p[A_HOR_R] != p[0,0,0,0,0,0]):
                $ 1099 "for_z_VR1≔A_Touch_p[A_HOR_R]"
                global for_z_VR1=A_Touch_p[A_HOR_R]
              end
              $ 1100 "If for_z_VR1≠p[0,0,0,0,0,0]"
              if (for_z_VR1 != p[0,0,0,0,0,0]):
                $ 1101 "z_diff≔get_feature_pose(for_z_VR1,A_Touch_p[A_VR1])"
                global z_diff=get_feature_pose(for_z_VR1,A_Touch_p[A_VR1])
                $ 1102 "A_Touch_p[A_VR1]=pose_trans(A_Touch_p[A_VR1], p[z_diff[0],0,0,0,0,0])"
                A_Touch_p[A_VR1]= pose_trans (A_Touch_p[A_VR1], p[z_diff[0],0,0,0,0,0])
              end
              $ 1103 "If b1_cell_info_R≟B or b1_cell_info_R≟D or b1_cell_info_R≟d or b1_cell_info_R≟E or b1_cell_info_R≟e"
              if (b1_cell_info_R == B  or  b1_cell_info_R == D  or  b1_cell_info_R == d  or  b1_cell_info_R == E  or  b1_cell_info_R == e):
                $ 1104 "A_Touch_p[A_VR1]=pose_trans(A_Touch_p[A_VR1], p[vert_scallup_r/1000,0,0,0,0,0])"
                A_Touch_p[A_VR1]= pose_trans (A_Touch_p[A_VR1], p[vert_scallup_r/1000,0,0,0,0,0])
              end
            end
            $ 1106 "A_Touch_p[A_VR1]=pose_trans(A_Touch_p[A_VR1], p[offset_3f_begin/1000,0,0,0,0,0])"
            A_Touch_p[A_VR1]= pose_trans (A_Touch_p[A_VR1], p[offset_3f_begin/1000,0,0,0,0,0])
          end
          $ 1107 "VR2"
          $ 1108 "If A_Prepos_l[A_VR2]≠p[0,0,0,0,0,0]"
          if (A_Prepos_l[A_VR2] != p[0,0,0,0,0,0]):
            $ 1109 "If b1_cell_info_R≟A or b1_cell_info_R≟C or b1_cell_info_R≟c or b1_cell_info_R≟D or b1_cell_info_R≟d or b1_cell_info_R≟E"
            if (b1_cell_info_R == A  or  b1_cell_info_R == C  or  b1_cell_info_R == c  or  b1_cell_info_R == D  or  b1_cell_info_R == d  or  b1_cell_info_R == E):
              $ 1110 "'3f only does not apply offset'"
              # '3f only does not apply offset'
              $ 1111 "If for_z_VLR2≟p[0,0,0,0,0,0] and A_Touch_p[A_HOR_MR]≠p[0,0,0,0,0,0]"
              if (for_z_VLR2 == p[0,0,0,0,0,0]  and  A_Touch_p[A_HOR_MR] != p[0,0,0,0,0,0]):
                $ 1112 "for_z_VLR2≔A_Touch_p[A_HOR_MR]"
                global for_z_VLR2=A_Touch_p[A_HOR_MR]
              end
              $ 1113 "Comment"
              # Comment
              $ 1114 "If for_z_VLR2≠p[0,0,0,0,0,0]"
              if (for_z_VLR2 != p[0,0,0,0,0,0]):
                $ 1115 "z_diff≔get_feature_pose(for_z_VLR2,A_Touch_p[A_VR2])"
                global z_diff=get_feature_pose(for_z_VLR2,A_Touch_p[A_VR2])
                $ 1116 "A_Touch_p[A_VR2]=pose_trans(A_Touch_p[A_VR2], p[z_diff[0],0,0,0,0,0])"
                A_Touch_p[A_VR2]= pose_trans (A_Touch_p[A_VR2], p[z_diff[0],0,0,0,0,0])
              end
              $ 1117 "If b1_cell_info_R≟E or b1_cell_info_R≟e"
              if (b1_cell_info_R == E  or  b1_cell_info_R == e):
                $ 1118 "A_Touch_p[A_VR2]=pose_trans(A_Touch_p[A_VR2], p[vert_scallup_r/1000,0,0,0,0,0])"
                A_Touch_p[A_VR2]= pose_trans (A_Touch_p[A_VR2], p[vert_scallup_r/1000,0,0,0,0,0])
              end
            end
            $ 1119 "A_Touch_p[A_VR2]=pose_trans(A_Touch_p[A_VR2], p[offset_3f_begin/1000,0,0,0,0,0])"
            A_Touch_p[A_VR2]= pose_trans (A_Touch_p[A_VR2], p[offset_3f_begin/1000,0,0,0,0,0])
          end
          $ 1120 "HOR_ML"
          $ 1121 "If A_Prepos_l[A_HOR_ML]≠p[0,0,0,0,0,0]"
          if (A_Prepos_l[A_HOR_ML] != p[0,0,0,0,0,0]):
            $ 1122 "A_Touch_p[A_HOR_M]=A_Touch_p[A_HOR_ML]"
            A_Touch_p[A_HOR_M]=A_Touch_p[A_HOR_ML]
            $ 1123 "x_welding_axis≔get_feature_pose(for_cal_x_wel,A_Touch_p[A_HOR_ML])"
            global x_welding_axis=get_feature_pose(for_cal_x_wel,A_Touch_p[A_HOR_ML])
            $ 1124 "A_Touch_p[A_HOR_M]=pose_trans(A_Touch_p[A_HOR_ML], p[x_welding_axis[0],0,0,0,0,0])"
            A_Touch_p[A_HOR_M]= pose_trans (A_Touch_p[A_HOR_ML], p[x_welding_axis[0],0,0,0,0,0])
            $ 1125 "A_Touch_p[A_HOR_M]=put_pose(A_Touch_p[A_HOR_M],0,for_cal_y_wel[0])"
            A_Touch_p[A_HOR_M]=put_pose(A_Touch_p[A_HOR_M],0,for_cal_y_wel[0])
            $ 1126 "A_Touch_p[A_HOR_M]=pose_trans(A_Touch_p[A_HOR_M], p[10/1000,0,0,0,0,0])"
            A_Touch_p[A_HOR_M]= pose_trans (A_Touch_p[A_HOR_M], p[10/1000,0,0,0,0,0])
            $ 1127 "If b1_cell_info_L≟C or b1_cell_info_L≟D"
            if (b1_cell_info_L == C  or  b1_cell_info_L == D):
              $ 1129 "x_welding_axis≔get_feature_pose(for_cal_x_wel,A_Touch_p[A_HOR_ML])"
              global x_welding_axis=get_feature_pose(for_cal_x_wel,A_Touch_p[A_HOR_ML])
              $ 1130 "A_Touch_p[A_HOR_ML]=pose_trans(A_Touch_p[A_HOR_ML],p[x_welding_axis[0],0,0,0,0,0])"
              A_Touch_p[A_HOR_ML]= pose_trans (A_Touch_p[A_HOR_ML],p[x_welding_axis[0],0,0,0,0,0])
              $ 1131 "A_Touch_p[A_HOR_ML]=pose_trans(A_Touch_p[A_HOR_ML],p[0/1000,0,0,0,0,0])"
              A_Touch_p[A_HOR_ML]= pose_trans (A_Touch_p[A_HOR_ML],p[0/1000,0,0,0,0,0])
            end
          end
          $ 1132 "HOR_MR"
          $ 1133 "If A_Prepos_l[A_HOR_MR]≠p[0,0,0,0,0,0]"
          if (A_Prepos_l[A_HOR_MR] != p[0,0,0,0,0,0]):
            $ 1135 "A_Touch_p[A_HOR_M]=A_Touch_p[A_HOR_MR]"
            A_Touch_p[A_HOR_M]=A_Touch_p[A_HOR_MR]
            $ 1136 "x_welding_axis≔get_feature_pose(for_cal_x_wel,A_Touch_p[A_HOR_MR])"
            global x_welding_axis=get_feature_pose(for_cal_x_wel,A_Touch_p[A_HOR_MR])
            $ 1137 "A_Touch_p[A_HOR_M]=pose_trans(A_Touch_p[A_HOR_M], p[x_welding_axis[0],0,0,0,0,0])"
            A_Touch_p[A_HOR_M]= pose_trans (A_Touch_p[A_HOR_M], p[x_welding_axis[0],0,0,0,0,0])
            $ 1138 "A_Touch_p[A_HOR_M]=put_pose(A_Touch_p[A_HOR_M],0,for_cal_y_wel[0])"
            A_Touch_p[A_HOR_M]=put_pose(A_Touch_p[A_HOR_M],0,for_cal_y_wel[0])
            $ 1139 "A_Touch_p[A_HOR_M]=pose_trans(A_Touch_p[A_HOR_M], p[-10/1000,0,0,0,0,0])"
            A_Touch_p[A_HOR_M]= pose_trans (A_Touch_p[A_HOR_M], p[-10/1000,0,0,0,0,0])
            $ 1140 "If b1_cell_info_R≟C or b1_cell_info_R≟D"
            if (b1_cell_info_R == C  or  b1_cell_info_R == D):
              $ 1142 "x_welding_axis≔get_feature_pose(for_cal_x_wel,A_Touch_p[A_HOR_MR])"
              global x_welding_axis=get_feature_pose(for_cal_x_wel,A_Touch_p[A_HOR_MR])
              $ 1143 "A_Touch_p[A_HOR_MR]=pose_trans(A_Touch_p[A_HOR_MR],p[x_welding_axis[0],0,0,0,0,0])"
              A_Touch_p[A_HOR_MR]= pose_trans (A_Touch_p[A_HOR_MR],p[x_welding_axis[0],0,0,0,0,0])
              $ 1144 "A_Touch_p[A_HOR_MR]=pose_trans(A_Touch_p[A_HOR_MR],p[-0/1000,0,0,0,0,0])"
              A_Touch_p[A_HOR_MR]= pose_trans (A_Touch_p[A_HOR_MR],p[-0/1000,0,0,0,0,0])
            end
          end
          $ 1145 "'Touch Remember On/OFF'"
          # 'Touch Remember On/OFF'
          $ 1146 "write_port_register(180,1)"
          write_port_register(180,1)
        else:
          $ 1147 "Else" "noBreak"
          $ 1148 "Ignore Touch and check error"
          $ 1149 "Auto_cur_cell≔0"
          global Auto_cur_cell=0
          $ 1150 "Loop Auto_cur_cell<Auto_total_cell"
          while (Auto_cur_cell<Auto_total_cell):
            $ 1151 "A_sel_v≔Auto_W_num[Auto_cur_cell]"
            global A_sel_v=Auto_W_num[Auto_cur_cell]
            $ 1152 "If A_sel_v<A_HOR_2path"
            if (A_sel_v<A_HOR_2path):
              $ 1153 "If A_Touch_p[A_sel_v]≟p[0,0,0,0,0,0]"
              if (A_Touch_p[A_sel_v] == p[0,0,0,0,0,0]):
                $ 1154 "write_port_register(142,120)"
                write_port_register(142,120)
                $ 1155 "Halt"
                halt
              end
            end
            $ 1156 "Auto_cur_cell≔Auto_cur_cell+1"
            global Auto_cur_cell=Auto_cur_cell+1
          end
          $ 1157 "Auto_cur_cell≔0"
          global Auto_cur_cell=0
        end
        $ 1158 "welding"
        $ 1159 "weldings"
        $ 1160 "Auto_cur_cell≔read_port_register(138)"
        global Auto_cur_cell= read_port_register (138)
        $ 1161 "time_cal_trig≔ True "
        global time_cal_trig=  True
        $ 1162 "Loop Auto_cur_cell<Auto_total_cell"
        while (Auto_cur_cell<Auto_total_cell):
          $ 1163 "write_port_register(138,Auto_cur_cell)"
          write_port_register(138,Auto_cur_cell)
          $ 1164 "running_trig≔ True "
          global running_trig=  True
          $ 1165 "'[2F_AB - 30] , [2F_CD_LEFT - 100] , [2F_CD_RIGHT - 150] , [3F - ELSE]'"
          # '[2F_AB - 30] , [2F_CD_LEFT - 100] , [2F_CD_RIGHT - 150] , [3F - ELSE]'
          $ 1166 "If Auto_W_num[Auto_cur_cell]≥100 and Auto_W_num[Auto_cur_cell]≤149"
          if (Auto_W_num[Auto_cur_cell] >= 100  and  Auto_W_num[Auto_cur_cell] <= 149):
            $ 1167 "'2F CD LEFT'"
            # '2F CD LEFT'
            $ 1168 "A_sel_v≔A_HOR"
            global A_sel_v=A_HOR
            $ 1169 "A_sel_v_end≔A_HOR_ML"
            global A_sel_v_end=A_HOR_ML
            $ 1170 "A_sel_v2≔A_HOR_M"
            global A_sel_v2=A_HOR_M
            $ 1171 "A_sel_v_end2≔A_HOR_R"
            global A_sel_v_end2=A_HOR_R
            $ 1172 "If floor(Auto_W_num[Auto_cur_cell]/10)≟10"
            if (floor(Auto_W_num[Auto_cur_cell]/10) == 10):
              $ 1173 "current_path≔1"
              global current_path=1
              $ 1174 "multi_path≔1"
              global multi_path=1
            else:
              $ 1175 "ElseIf floor(Auto_W_num[Auto_cur_cell]/10)≟11"
              if (floor(Auto_W_num[Auto_cur_cell]/10) == 11):
                $ 1176 "current_path≔2"
                global current_path=2
                $ 1177 "multi_path≔2"
                global multi_path=2
              else:
                $ 1178 "ElseIf floor(Auto_W_num[Auto_cur_cell]/10)≟12"
                if (floor(Auto_W_num[Auto_cur_cell]/10) == 12):
                  $ 1179 "current_path≔3"
                  global current_path=3
                  $ 1180 "multi_path≔3"
                  global multi_path=3
                else:
                  $ 1181 "ElseIf floor(Auto_W_num[Auto_cur_cell]/10)≟13"
                  if (floor(Auto_W_num[Auto_cur_cell]/10) == 13):
                    $ 1182 "current_path≔4"
                    global current_path=4
                    $ 1183 "multi_path≔4"
                    global multi_path=4
                  end
                end
              end
            end
            $ 1184 "current_2f≔current_2f+1"
            global current_2f=current_2f+1
            $ 1185 "CD_MLR≔ True "
            global CD_MLR=  True
            $ 1186 "write_port_register(135,A_HOR)"
            write_port_register(135,A_HOR)
            $ 1187 "write_port_register(136,current_2f)"
            write_port_register(136,current_2f)
            $ 1188 "If simulation_mode"
            if (simulation_mode):
              $ 1189 "Call welding_parameter_sim"
              welding_parameter_sim()
            else:
              $ 1190 "Else" "noBreak"
              $ 1191 "Call welding_parameter_init"
              welding_parameter_init()
            end
            $ 1192 "wv_direction≔1"
            global wv_direction=1
            $ 1193 "If Auto_W_num[Auto_cur_cell]%10≟4"
            if (Auto_W_num[Auto_cur_cell]%10 == 4):
              $ 1194 "A_sel_v≔A_HOR_R"
              global A_sel_v=A_HOR_R
              $ 1195 "Call MoveFun"
              MoveFun()
              $ 1196 "A_sel_v≔A_HOR"
              global A_sel_v=A_HOR
            else:
              $ 1197 "ElseIf Auto_W_num[Auto_cur_cell]%10≟0 or Auto_W_num[Auto_cur_cell]%10≟1 or Auto_W_num[Auto_cur_cell]%10≟2"
              if (Auto_W_num[Auto_cur_cell]%10 == 0  or  Auto_W_num[Auto_cur_cell]%10 == 1  or  Auto_W_num[Auto_cur_cell]%10 == 2):
                $ 1198 "Call MoveFun"
                MoveFun()
              end
            end
            $ 1199 "Call weav_welding_2f_CD"
            weav_welding_2f_CD()
          else:
            $ 1200 "ElseIf Auto_W_num[Auto_cur_cell]≥150 and Auto_W_num[Auto_cur_cell]≤189"
            if (Auto_W_num[Auto_cur_cell] >= 150  and  Auto_W_num[Auto_cur_cell] <= 189):
              $ 1201 "'2F CD RIGHT'"
              # '2F CD RIGHT'
              $ 1202 "A_sel_v≔A_HOR_R"
              global A_sel_v=A_HOR_R
              $ 1203 "A_sel_v_end≔A_HOR_MR"
              global A_sel_v_end=A_HOR_MR
              $ 1204 "A_sel_v2≔A_HOR_M"
              global A_sel_v2=A_HOR_M
              $ 1205 "A_sel_v_end2≔A_HOR"
              global A_sel_v_end2=A_HOR
              $ 1206 "If floor(Auto_W_num[Auto_cur_cell]/10)≟15"
              if (floor(Auto_W_num[Auto_cur_cell]/10) == 15):
                $ 1207 "current_path≔1"
                global current_path=1
                $ 1208 "multi_path≔1"
                global multi_path=1
              else:
                $ 1209 "ElseIf floor(Auto_W_num[Auto_cur_cell]/10)≟16"
                if (floor(Auto_W_num[Auto_cur_cell]/10) == 16):
                  $ 1210 "current_path≔2"
                  global current_path=2
                  $ 1211 "multi_path≔2"
                  global multi_path=2
                else:
                  $ 1212 "ElseIf floor(Auto_W_num[Auto_cur_cell]/10)≟17"
                  if (floor(Auto_W_num[Auto_cur_cell]/10) == 17):
                    $ 1213 "current_path≔3"
                    global current_path=3
                    $ 1214 "multi_path≔3"
                    global multi_path=3
                  else:
                    $ 1215 "ElseIf floor(Auto_W_num[Auto_cur_cell]/10)≟18"
                    if (floor(Auto_W_num[Auto_cur_cell]/10) == 18):
                      $ 1216 "current_path≔4"
                      global current_path=4
                      $ 1217 "multi_path≔4"
                      global multi_path=4
                    end
                  end
                end
              end
              $ 1218 "current_2f≔current_2f+1"
              global current_2f=current_2f+1
              $ 1219 "CD_MLR≔ False "
              global CD_MLR=  False
              $ 1220 "write_port_register(135,A_HOR)"
              write_port_register(135,A_HOR)
              $ 1221 "write_port_register(136,current_2f)"
              write_port_register(136,current_2f)
              $ 1222 "If simulation_mode"
              if (simulation_mode):
                $ 1223 "Call welding_parameter_sim"
                welding_parameter_sim()
              else:
                $ 1224 "Else" "noBreak"
                $ 1225 "Call welding_parameter_init"
                welding_parameter_init()
              end
              $ 1226 "wv_direction≔-1"
              global wv_direction=-1
              $ 1227 "If Auto_W_num[Auto_cur_cell]%10≟4"
              if (Auto_W_num[Auto_cur_cell]%10 == 4):
                $ 1228 "A_sel_v≔A_HOR"
                global A_sel_v=A_HOR
                $ 1229 "Call MoveFun"
                MoveFun()
                $ 1230 "A_sel_v≔A_HOR_R"
                global A_sel_v=A_HOR_R
              else:
                $ 1231 "ElseIf Auto_W_num[Auto_cur_cell]%10≟0 or Auto_W_num[Auto_cur_cell]%10≟1 or Auto_W_num[Auto_cur_cell]%10≟2"
                if (Auto_W_num[Auto_cur_cell]%10 == 0  or  Auto_W_num[Auto_cur_cell]%10 == 1  or  Auto_W_num[Auto_cur_cell]%10 == 2):
                  $ 1232 "Call MoveFun"
                  MoveFun()
                end
              end
              $ 1233 "Call weav_welding_2f_CD"
              weav_welding_2f_CD()
            else:
              $ 1234 "ElseIf Auto_W_num[Auto_cur_cell]≥30 and Auto_W_num[Auto_cur_cell]≤65"
              if (Auto_W_num[Auto_cur_cell] >= 30  and  Auto_W_num[Auto_cur_cell] <= 65):
                $ 1235 "'2F'"
                # '2F'
                $ 1236 "A_sel_v≔A_HOR"
                global A_sel_v=A_HOR
                $ 1237 "A_sel_v_end≔A_HOR_R"
                global A_sel_v_end=A_HOR_R
                $ 1238 "If floor(Auto_W_num[Auto_cur_cell]/10)≟3"
                if (floor(Auto_W_num[Auto_cur_cell]/10) == 3):
                  $ 1239 "current_path≔1"
                  global current_path=1
                  $ 1240 "multi_path≔1"
                  global multi_path=1
                else:
                  $ 1241 "ElseIf floor(Auto_W_num[Auto_cur_cell]/10)≟4"
                  if (floor(Auto_W_num[Auto_cur_cell]/10) == 4):
                    $ 1242 "current_path≔2"
                    global current_path=2
                    $ 1243 "multi_path≔2"
                    global multi_path=2
                  else:
                    $ 1244 "ElseIf floor(Auto_W_num[Auto_cur_cell]/10)≟5"
                    if (floor(Auto_W_num[Auto_cur_cell]/10) == 5):
                      $ 1245 "current_path≔3"
                      global current_path=3
                      $ 1246 "multi_path≔3"
                      global multi_path=3
                    else:
                      $ 1247 "ElseIf floor(Auto_W_num[Auto_cur_cell]/10)≟6"
                      if (floor(Auto_W_num[Auto_cur_cell]/10) == 6):
                        $ 1248 "current_path≔4"
                        global current_path=4
                        $ 1249 "multi_path≔4"
                        global multi_path=4
                      end
                    end
                  end
                end
                $ 1250 "current_2f≔current_2f+1"
                global current_2f=current_2f+1
                $ 1251 "write_port_register(135,A_HOR)"
                write_port_register(135,A_HOR)
                $ 1252 "write_port_register(136,current_2f)"
                write_port_register(136,current_2f)
                $ 1253 "If simulation_mode"
                if (simulation_mode):
                  $ 1254 "Call welding_parameter_sim"
                  welding_parameter_sim()
                else:
                  $ 1255 "Else" "noBreak"
                  $ 1256 "Call welding_parameter_init"
                  welding_parameter_init()
                end
                $ 1257 "If Auto_W_num[Auto_cur_cell]%10≟2"
                if (Auto_W_num[Auto_cur_cell]%10 == 2):
                  $ 1258 "A_sel_v≔A_HOR_R"
                  global A_sel_v=A_HOR_R
                  $ 1259 "Call MoveFun"
                  MoveFun()
                  $ 1260 "A_sel_v≔A_HOR"
                  global A_sel_v=A_HOR
                else:
                  $ 1261 "Else" "noBreak"
                  $ 1262 "Call MoveFun"
                  MoveFun()
                end
                $ 1263 "Call weav_welding_2f"
                weav_welding_2f()
              else:
                $ 1264 "Else" "noBreak"
                $ 1265 "A_sel_v≔Auto_W_num[Auto_cur_cell]"
                global A_sel_v=Auto_W_num[Auto_cur_cell]
                $ 1266 "write_port_register(135,A_sel_v)"
                write_port_register(135,A_sel_v)
                $ 1267 "current_path≔1"
                global current_path=1
                $ 1268 "current_2f≔0"
                global current_2f=0
                $ 1269 "write_port_register(136,current_2f)"
                write_port_register(136,current_2f)
                $ 1270 "If simulation_mode"
                if (simulation_mode):
                  $ 1271 "Call welding_parameter_sim"
                  welding_parameter_sim()
                else:
                  $ 1272 "Else" "noBreak"
                  $ 1273 "Call welding_parameter_init"
                  welding_parameter_init()
                end
                $ 1274 "A_sel_v_end≔A_sel_v+9"
                global A_sel_v_end=A_sel_v+9
                $ 1275 "Call weav_welding_3f"
                weav_welding_3f()
              end
            end
          end
          $ 1276 "Call reset_weld_param"
          reset_weld_param()
          $ 1277 "next_before"
          $ 1278 "If get_move_trig≟1"
          if (get_move_trig == 1):
            $ 1279 "If get_next_number≠Auto_cur_cell"
            if (get_next_number != Auto_cur_cell):
              $ 1280 "Auto_cur_cell≔get_next_number"
              global Auto_cur_cell=get_next_number
            else:
              $ 1281 "Else" "noBreak"
              $ 1282 "Auto_cur_cell≔Auto_cur_cell+1"
              global Auto_cur_cell=Auto_cur_cell+1
            end
            $ 1283 "write_port_register(166,0)"
            write_port_register(166,0)
            $ 1284 "write_port_register(167,0)"
            write_port_register(167,0)
            $ 1285 "get_move_trig≔0"
            global get_move_trig=0
          else:
            $ 1286 "Else" "noBreak"
            $ 1287 "Auto_cur_cell≔Auto_cur_cell+1"
            global Auto_cur_cell=Auto_cur_cell+1
          end
        end
        $ 1288 "homeing()"
        homeing()
        $ 1289 "write_port_register(162,1)"
        write_port_register(162,1)
        $ 1290 "write_port_register(180,0)"
        write_port_register(180,0)
        thread_flag_306 = 1
      end
      if (a0_Job_Mode == 2):
        global thread_handler_306=run Thread_if_306()
        while (thread_flag_306 == 0):
          if not(a0_Job_Mode == 2):
            kill thread_handler_306
            thread_flag_306 = 2
          else:
            sync()
          end
        end
      else:
        thread_flag_306 = 2
      end
    end
    $ 1291 "Wait: 0.01"
    sleep(0.01)
    $ 1292 "after init auto"
    $ 1293 "If auto_on"
    if (auto_on):
      $ 1294 "write_port_register(202,0)"
      write_port_register(202,0)
      $ 1295 "timer_1: Stop"
      timer_1_is_counting = False
      $ 1296 "write_welder(0, False )"
      write_welder(0,  False  )
      $ 1297 "write_welder(4, False )"
      write_welder(4,  False  )
      $ 1298 "Call reset_weld_param"
      reset_weld_param()
      $ 1299 "Call reset_multi_record"
      reset_multi_record()
      $ 1300 "multi_path≔1"
      global multi_path=1
      $ 1301 "auto_on≔ False "
      global auto_on=  False
      $ 1302 "current_2f≔0"
      global current_2f=0
      $ 1303 "get_center≔get_center_bak"
      global get_center=get_center_bak
      $ 1304 "vr2_p1≔p[0,0,0,0,0,0]"
      global vr2_p1=p[0,0,0,0,0,0]
      $ 1305 "welding_program≔ False "
      global welding_program=  False
      $ 1306 "start_num≔135"
      global start_num=135
      $ 1307 "Loop start_num<141"
      while (start_num<141):
        $ 1308 "write_port_register(start_num,0)"
        write_port_register(start_num,0)
        $ 1309 "start_num≔start_num+1"
        global start_num=start_num+1
      end
    end
  end
end
